Yaskawa INFORM job: R1_W70(-90,-90)KM-OK.JBI

/JOB
//NAME R1_W70(-90,-90)KM-OK
///FOLDERNAME KRIS-SCIANA
//POS
///NPOS 26,26,0,2,0,0
///TOOL 0
///POSTYPE PULSE
///PULSE
C00000=196132,-11386,-19710,25477,112172,-12618
C00001=198011,-10737,-15790,25505,109711,-12435
C00002=198761,-10389,-14149,25526,108727,-12362
C00003=197276,-7784,-9608,24959,107857,-13151
C00004=197885,-8427,-9274,25015,107185,-13060
C00005=197276,-7784,-9608,24959,107857,-13151
C00006=198761,-10389,-14149,25526,108727,-12362
C00007=193286,-15234,-12496,33984,104867,-14280
C00008=192731,-14102,-10699,33783,104648,-14584
C00009=193286,-15234,-12496,33984,104867,-14280
C00010=191707,-13721,-12199,33776,105994,-14592
C00011=204462,-14015,-20466,16962,112467,-10975
C00012=206397,-15409,-17654,17145,109719,-10647
C00013=206838,-13484,-16187,17267,109709,-10480
C00014=206397,-15409,-17654,17145,109719,-10647
C00015=200372,-42268,-41130,22283,97203,-14677
C00016=196030,-47761,-46906,25813,86896,59583
C00017=191753,-49185,-38178,35401,78810,66101
C00018=192636,-50532,-38220,35397,77895,66172
C00019=192317,-49774,-38245,35380,78361,66190
C00020=191548,-48654,-37176,35452,78613,65950
C00021=192854,-50154,-37695,35384,77693,66198
C00022=197654,-39269,-30814,34764,76845,67931
C00023=190949,-52971,-46379,35207,81700,66696
C00024=185515,-45379,-43888,35551,85902,65801
C00025=121469,-120277,-97944,10587,51234,-59350
BC00000=387107,1191142,1068222
BC00001=387107,1191142,1068222
BC00002=387107,1191142,1068222
BC00003=387107,1191142,1068222
BC00004=387107,1191142,1068222
BC00005=387107,1191142,1068222
BC00006=387107,1191142,1068222
BC00007=387107,1191142,1068222
BC00008=387107,1191142,1068222
BC00009=387107,1191142,1068222
BC00010=387107,1191142,1068222
BC00011=387107,1191142,1068222
BC00012=387107,1191142,1068222
BC00013=387107,1191142,1068222
BC00014=387107,1191142,1068222
BC00015=387107,1191142,1068222
BC00016=387107,1191142,1068222
BC00017=386184,1191142,1068222
BC00018=385923,1191142,1068222
BC00019=385923,1191142,1068222
BC00020=385923,1191142,1068222
BC00021=382378,1191142,1068222
BC00022=377600,1191142,1068222
BC00023=377861,1191142,1068222
BC00024=377861,1191142,1068222
BC00025=220393,1191142,1068222
///POSTYPE BASE
///RECTAN
///RCONF 0,0,0,0,0,0,0,0,0,0,0,0,0,0,0,0,0,0,0,0,0,0,0,0
P00006=0.222,-3.123,-1.508,0.0000,0.0000,0.0000
P00022=0.222,-3.123,-1.508,0.0000,0.0000,0.0000
//INST
///DATE 2024/07/23 16:14
///ATTR SC,RW
///GROUP1 RB1,BS1
NOP
'r1_W70(-90,-90)
'Path S890
SFTOF
MOVJ C00000 BC00000 VJ=20.00
MOVJ C00001 BC00001 VJ=20.00
MOVL C00002 BC00002 V=100.0
MOVL C00003 BC00003 V=60.0
REFP 3 C00004 BC00004
CALL JOB:SEARCH-R1
SET P022 P006
SFTON P022
MOVL C00005 BC00005 V=60.0
MOVL C00006 BC00006 V=100.0
MOVL C00007 BC00007 V=60.0
REFP 3 C00008 BC00008
CALL JOB:SEARCH-R1
SET P022 P006
SFTON P022
MOVL C00009 BC00009 V=60.0
MOVL C00010 BC00010 V=100.0
MOVL C00011 BC00011 V=100.0
MOVL C00012 BC00012 V=60.0
REFP 3 C00013 BC00013
CALL JOB:SEARCH-R1
SET P022 P006
SFTON P022
MOVL C00014 BC00014 V=60.0
MOVL C00015 BC00015 V=100.0
MOVL C00016 BC00016 V=100.0
'Path W509
SFTOF
SFTON P022
MOVJ C00017 BC00017 VJ=20.00
MOVL C00018 BC00018 V=166.7 PL=0
REFP 1 C00019 BC00019
REFP 2 C00020 BC00020
MACRO1 MJ#(0) ARGF7
ARCON
MOVL C00021 BC00021 V=10.0
MOVL C00022 BC00022 V=10.0
ARCOF
MOVL C00023 BC00023 V=166.7
MOVJ C00024 BC00024 VJ=100.00
SFTOF
MOVJ C00025 BC00025 VJ=100.00
END
